FUNCTION_BLOCK ClimatSystem EXTENDS Device IMPLEMENTS SHLib.IInputDevice, SHLib.IOutputDevice
VAR
	_Temperature : SINT := 25;
	
	_IsCoolingOn : BOOL;
	_IsHeatingOn : BOOL;
END_VAR

{attribute 'monitoring' := 'call'}
PROPERTY IsCoolingOn : BOOL
GET
IsCoolingOn := _IsCoolingOn;
END_GET
END_PROPERTY

{attribute 'monitoring' := 'call'}
PROPERTY IsHeatingOn : BOOL
GET
IsHeatingOn := _IsHeatingOn;
END_GET
END_PROPERTY

{attribute 'monitoring' := 'call'}
PROPERTY Name : STRING
GET
Name := 'ClimatSystem';
END_GET
END_PROPERTY

METHOD ReadInputs
// handle value from terminal here
END_METHOD

{attribute 'monitoring' := 'call'}
PROPERTY Temperature : SINT
GET
Temperature := _Temperature;
END_GET
END_PROPERTY

METHOD WriteOutputs
_IsHeatingOn := _Temperature <= 20;
_IsCoolingOn := _Temperature >= 30;
END_METHOD

END_FUNCTION_BLOCK

(* stored: Version 1.1.0.1
   POU ClimatSystem: Id {d5c9f4d7-442e-4350-b38e-72270214942d}, SpecialFunc None
   Property IsCoolingOn: Id {5b45d383-5f49-4517-a50f-625530fae5ce}
   Get Get: Id {5f83f3cc-2dc6-44d0-a203-f1c8b48a1525}
   Property IsHeatingOn: Id {828ee96e-21b4-4e34-806a-543797de5bbf}
   Get Get: Id {ce639004-d103-47c0-9902-eb26fcb07b0d}
   Property Name: Id {6b9ccc29-dfff-4927-81ce-27cbd43db212}
   Get Get: Id {9f9b7976-f60d-43b4-a92f-220a5c8e3fc5}
   Method ReadInputs: Id {befd84e7-279d-42f9-bcb3-cd989af07b0f}
   Property Temperature: Id {10cfe9f1-989b-4b93-93ac-40dff08806b8}
   Get Get: Id {3cffbb6f-ab2f-4faa-a477-6d68b2e7bd67}
   Method WriteOutputs: Id {e7fe7906-23f2-4f3e-9cca-ab9f37a2f9b9} *)
